TYPE ST_Nest :
STRUCT
    nId                       : UINT;
    ePosition                 : E_TablePosition;
    bEnabled                  : BOOL;
    bPartPresent              : BOOL;
    bPreviousPartPresent      : BOOL;
    bPartLoadedPulse          : BOOL;
    bPartRemovedPulse         : BOOL;
    bProcessRequired          : BOOL;
    bProcessComplete          : BOOL;
    eDisposition              : E_PartDisposition;
    bDispositionSent          : BOOL;
    bOperatorExchangeComplete : BOOL;
    stPatchDispenseResult     : ST_ProcessResult;
    stHeatStakeResult         : ST_ProcessResult;
    stVisionResult            : ST_ProcessResult;

    ePatchDispenseStage       : E_NestStageStatus := E_NestStageStatus.Waiting;
    eHeatStakeStage           : E_NestStageStatus := E_NestStageStatus.Waiting;
    eVisionStage              : E_NestStageStatus := E_NestStageStatus.Waiting;

    stResult                  : ST_ProcessResult;
    bStatisticsCounted        : BOOL;
    // Live at Operator / last observed off Operator; bPartPresent remains PRODUCT only.
    bPbupPresent : BOOL;
    // Historical paired load for this product; not invalidated by PBUP assembly at Vision.
    bLoadSetComplete : BOOL;
END_STRUCT
END_TYPE

(* stored: Version 1.1.0.1, ProductVersion 3.1.4026.18
   DUT ST_Nest: Id {e9c52966-abb7-45b8-ba6f-050cecbcb7e1} *)
